(* PLC project Untitled1, Beckhoff Automation GmbH TF6420 Database Server Query Analyser 1.0.0.0 *)
(* stored: creationDateTime 2018-09-28T13:19:20, modificationDateTime 2018-09-28T13:19:20 *)

TYPE ST_ProgramStruct : STRUCT
  ID : DINT;
  Time : DT;
  setpoint : REAL;
END_STRUCT;
END_TYPE
